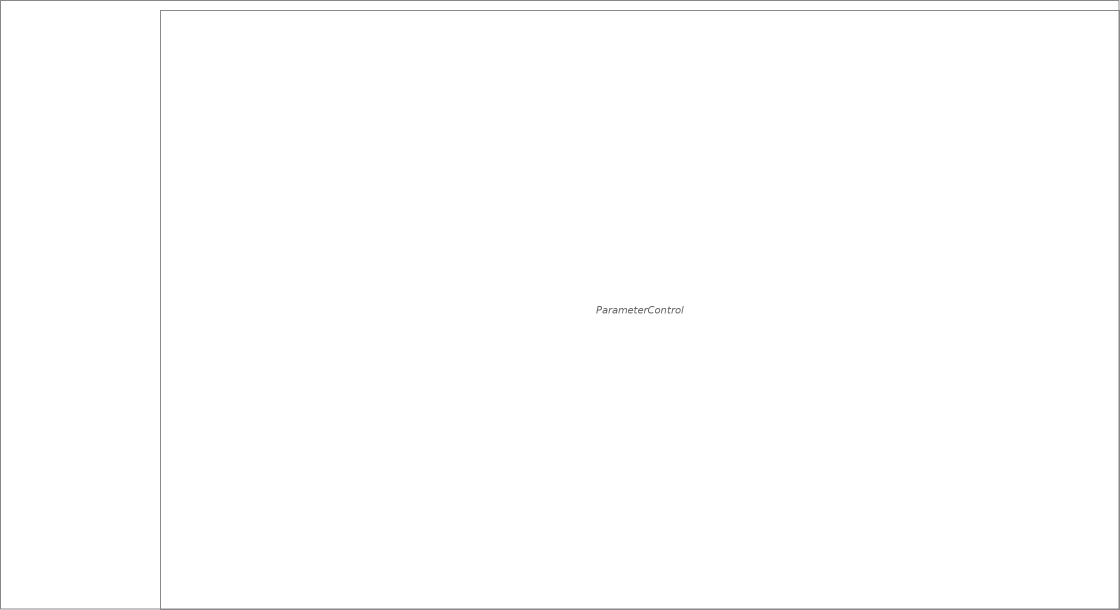
VISUALIZATION Parameters  // 1120x610
    Frame (160,10 960x600)
        shows ParameterControl()
END_VISUALIZATION

(* stored: Version 1.1.0.1, ProductVersion 3.1.4024.11
   Visu Parameters: Id {5868e799-14d6-48dd-8c7e-b96f37ed34ae} *)
